INTERFACE ITFPalletStacker

METHOD CollectPallet
VAR_INPUT
END_VAR
END_METHOD

METHOD EmptyStack
VAR_INPUT
END_VAR
END_METHOD

METHOD Reset
VAR_INPUT
END_VAR
END_METHOD

METHOD StackPallet
VAR_INPUT
END_VAR
END_METHOD

PROPERTY Status : E_DeviceStatus
GET
END_GET
SET
END_SET
END_PROPERTY

METHOD Stop
VAR_INPUT
END_VAR
END_METHOD

END_INTERFACE

(* stored: Version 1.1.0.1
   Itf ITFPalletStacker: Id {f1bf6491-f939-4a60-ac07-e60f6a94ec4e}
   Method CollectPallet: Id {42c406db-0f81-4711-818d-aef16ab72e5b}
   Method EmptyStack: Id {0ca567c3-45d2-4648-856b-671c4db26acb}
   Method Reset: Id {252bf8bf-c662-4138-ab5c-2fc71d5a722f}
   Method StackPallet: Id {0ce9402f-c1ee-4b57-83de-8b71bd4726d9}
   Property Status: Id {e47a648e-819f-4a16-8245-cbcff79a32bb}
   Get Get: Id {fefecf09-14e3-4783-945f-8b3c6f2e4eb4}
   Set Set: Id {b117357d-ebf8-4594-b05f-dcec9ef726c7}
   Method Stop: Id {86ff3a8b-19d4-4d1b-8aa5-453ade1e6d14} *)
